TYPE
    ST_FeedInEmptyBox_Status EXTENDS ST_StatusBasic :
    STRUCT
		
    END_STRUCT
END_TYPE

(* stored: Version 1.1.0.1, ProductVersion 3.1.4024.13
   DUT ST_FeedInEmptyBox_Status: Id {f1178e3d-788a-421b-96c7-db27ce346bcf} *)
